// TIA Portal V20 export
TYPE "typeSequenceControlNodeJobInterface"
// stored: Namespace Unit1.Em4
   STRUCT
      commands : "Unit1.Em4.typeSequenceControlNodeJobInterfaceCommands";
      monitoring { S7_SetPoint := 'True'} : "Unit1.Em4.typeSequenceControlNodeJobInterfaceMonitoring";
   END_STRUCT;
END_TYPE
